FUNCTION_BLOCK FB_UpdateTimeStamp
VAR_INPUT
END_VAR
VAR_OUTPUT
	FullSystemTime	: STRING;
	SystemDate		: STRING;
	SystemTime		: STRING;
	SystemHour		: STRING;
	timeValid		: bool;
END_VAR
VAR
	fb_LocalTime	 : FB_LocalSystemTime;
END_VAR

fb_LocalTime(
		sNetID:= , 
		bEnable:= TRUE , 
		dwCycle:= 1, 
		dwOpt:= , 
		tTimeout:= ,
		bValid=> timeValid, 
		systemTime=> , 
		tzID=> );
		
IF fb_localTime.bValid THEN
	FullSystemTime 	:= SYSTEMTIME_TO_STRING(fb_LocalTime.systemTime);
	
	SystemDate		:= WORD_TO_STRING(fb_LocalTime.systemTime.wYear);
	SystemDate		:= CONCAT(SystemDate, '.');
	SystemDate		:= CONCAT(SystemDate, WORD_TO_STRING(fb_LocalTime.systemTime.wMonth));
	SystemDate		:= CONCAT(SystemDate, '.');
	SystemDate		:= CONCAT(SystemDate, WORD_TO_STRING(fb_LocalTime.systemTime.wDay));
	
	SystemTime		:= WORD_TO_STRING(fb_LocalTime.systemTime.wHour);
	SystemTime		:= CONCAT(SystemTime, ':');
	SystemTime		:= CONCAT(SystemTime, WORD_TO_STRING(fb_LocalTime.systemTime.wMinute));
	SystemTime		:= CONCAT(SystemTime, ':');
	SystemTime		:= CONCAT(SystemTime, WORD_TO_STRING(fb_LocalTime.systemTime.wSecond));
	
	SystemHour		:= WORD_TO_STRING(fb_LocalTime.systemTime.wHour);
END_IF

END_FUNCTION_BLOCK

(* stored: Version 1.1.0.1, ProductVersion 3.1.4024.12
   POU FB_UpdateTimeStamp: Id {ae735186-4697-4995-bd8e-265b3602c2fb}, SpecialFunc None *)
